(* Schneider Machine Expert - Basic project usine, file version 2.8.0.0 *)
(* ProjectInformations: Name=Nouveau projet *)

HARDWARE
  Cpu 0: TM221M16R/G
  ModuleExtensionObject 0: TM3AQ4/G
  EthernetConfiguration: NetworkName=M221, IpAllocationMode=FixedAddress, IpAddress=0.0.0.0, SubnetMask=0.0.0.0
  SerialLineConfiguration: Baud=Baud19200, Parity=ParityEven, DataBits=DataBits8, StopBits=StopBits1, PhysicalMedium=PhysicalMediumRs485, TransmissionMode=TransmissionModeModbusRtu, SlaveId=1, Addressing=SlaveAddressing
  MastTask: UsePeriodScanMode=false, PeriodScan=100
  FastTask: Period=255
  CpuBehavior: StartingMode=StartAsPreviousState, AutoSaveRamOnEeprom=true, WatchdogPeriod=250

SYMBOLS  (address, symbol, comment, settings)
  %M0       M1
  %M1       M2
  %M3       LP
  %M4       SP
  %M5       TIME
  %M6       M
  %M7       H
  %M8       MODE_AUTO
  %M9       MARCHE_DES_MACHINE
  %M10      SS
  %S6       SB_TB1S  "Base de temps de 1 s générée par une horloge interne"
  %C0         [Preset=5]
  %C1         [Preset=5]
  %C2         [Preset=4]
  %I0.0     COURANT_M_1
  %I0.1     COURANT_M_2
  %I0.2     COURANT_M_3
  %I0.3     BP
  %I0.4     BP_MARCHE
  %I0.5     BP_STOP
  %I0.6     BP_AUTO
  %I0.7     BP_AUTO_S
  %Q0.0     MACHINE_R
  %Q0.1     MACHINE_B
  %Q0.2     MOTEUR

POU cable machine
  (* SectionNumber=1 *)

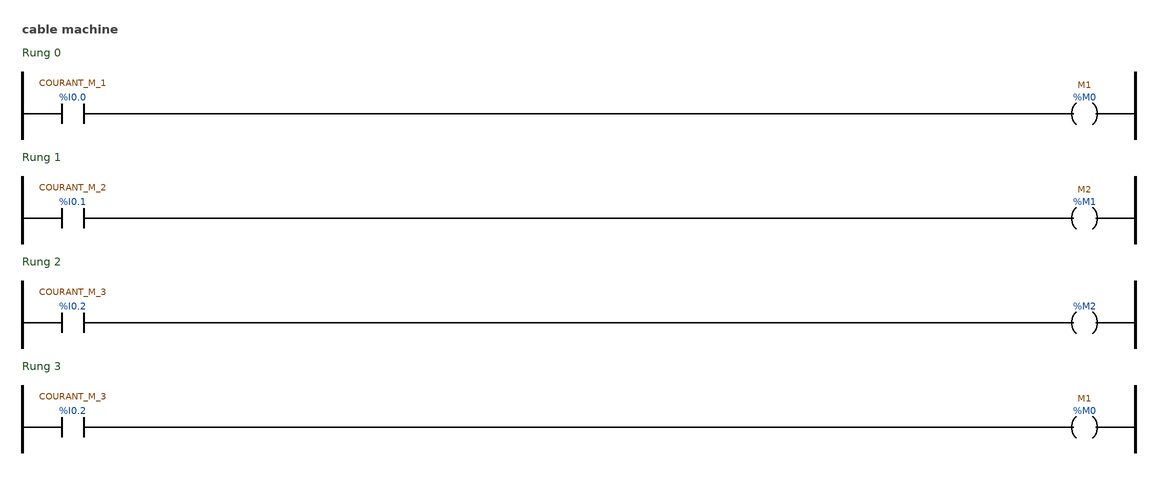

// Rung 0
  LD %I0.0                (* COURANT_M_1 *)
  ST %M0                  (* M1 *)
  // as ST:
  //   M1 := COURANT_M_1;

// Rung 1
  LD %I0.1                (* COURANT_M_2 *)
  ST %M1                  (* M2 *)
  // as ST:
  //   M2 := COURANT_M_2;

// Rung 2
  LD %I0.2                (* COURANT_M_3 *)
  ST %M2
  // as ST:
  //   %M2 := COURANT_M_3;

// Rung 3
  LD %I0.2                (* COURANT_M_3 *)
  ST %M0                  (* M1 *)
  // as ST:
  //   M1 := COURANT_M_3;

POU régulation
  (* SectionNumber=2 *)

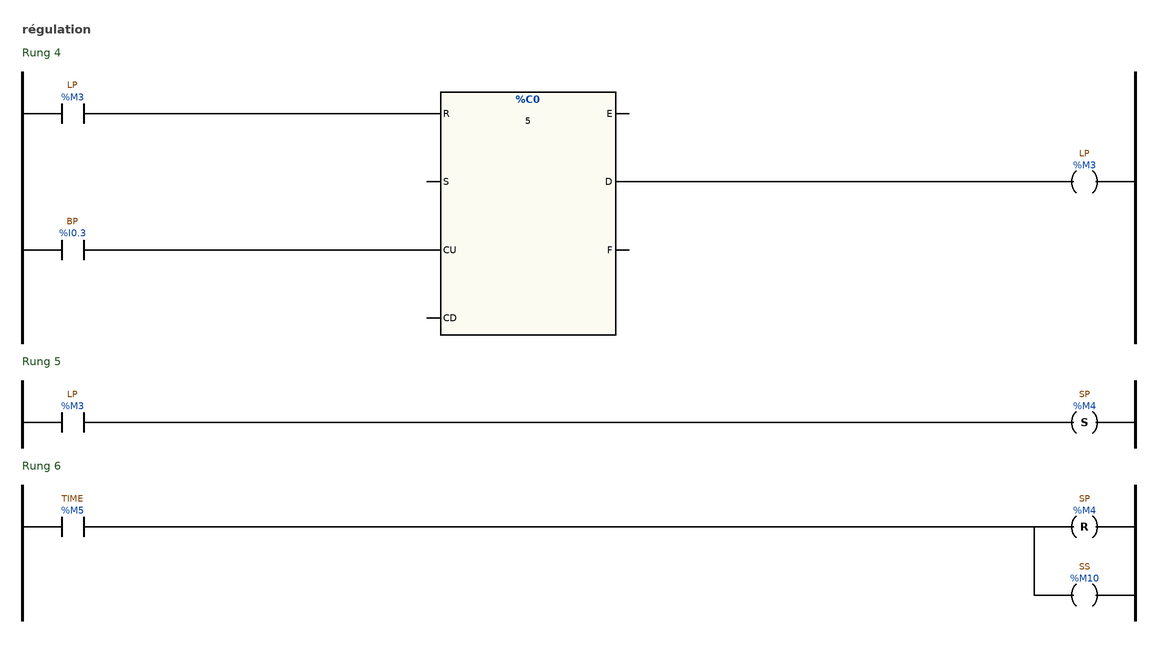

// Rung 4
  BLK %C0
  LD %M3                  (* LP *)
  R
  LD %I0.3                (* BP *)
  CU
  OUT_BLK
  LD D
  ST %M3                  (* LP *)
  END_BLK
  // as ST:
  //   %C0(R := LP, CU := BP);
  //   LP := %C0.D;

// Rung 5
  LD %M3                  (* LP *)
  S %M4                   (* SP *)
  // as ST:
  //   IF LP THEN SP := TRUE; END_IF;

// Rung 6
  LD %M5                  (* TIME *)
  R %M4                   (* SP *)
  ST %M10                 (* SS *)
  // as ST:
  //   IF TIME THEN SP := FALSE; END_IF;
  //   SS := TIME;

POU timer
  (* SectionNumber=3 *)

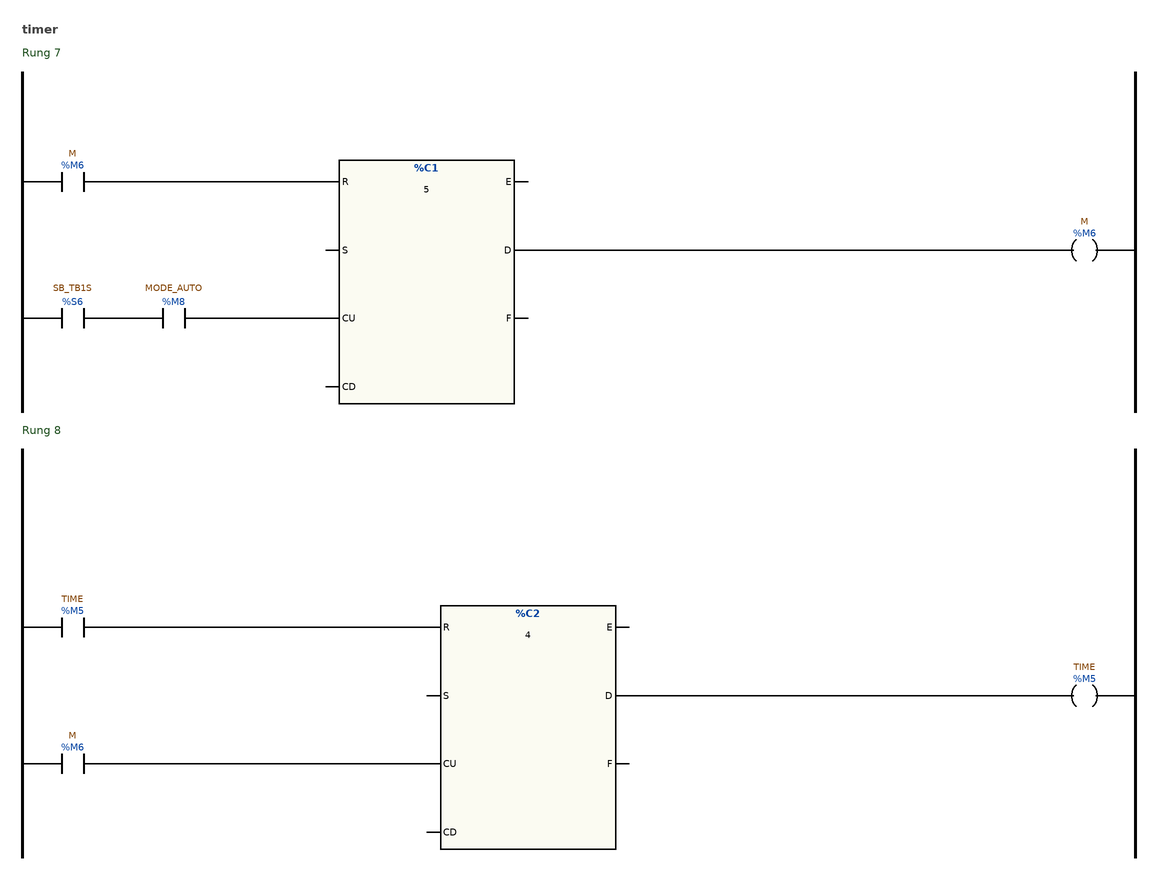

// Rung 7
  BLK %C1
  LD %M6                  (* M *)
  R
  LD %S6                  (* SB_TB1S *)
  AND %M8                 (* MODE_AUTO *)
  CU
  OUT_BLK
  LD D
  ST %M6                  (* M *)
  END_BLK
  // as ST:
  //   %C1(R := M, CU := SB_TB1S AND MODE_AUTO);
  //   M := %C1.D;

// Rung 8
  BLK %C2
  LD %M5                  (* TIME *)
  R
  LD %M6                  (* M *)
  CU
  OUT_BLK
  LD D
  ST %M5                  (* TIME *)
  END_BLK
  // as ST:
  //   %C2(R := TIME, CU := M);
  //   TIME := %C2.D;

POU start machine
  (* SectionNumber=4 *)

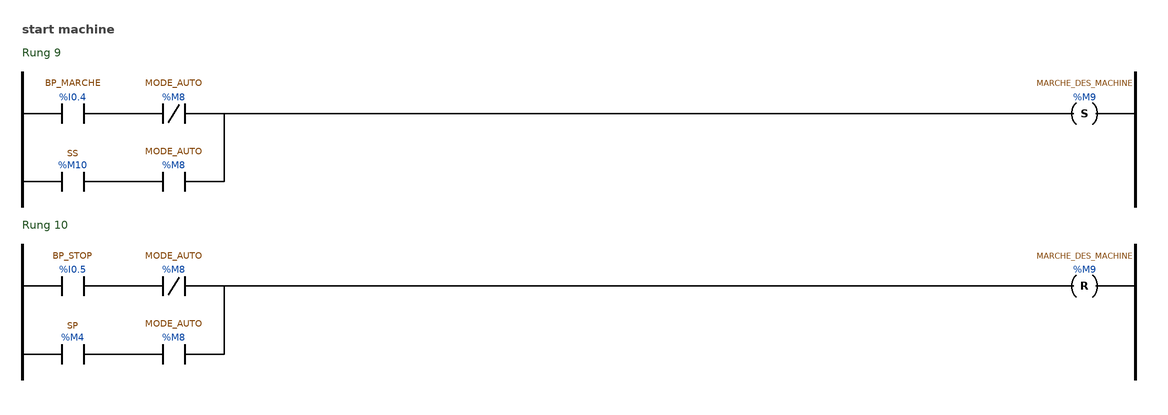

// Rung 9
  LD %I0.4                (* BP_MARCHE *)
  ANDN %M8                (* MODE_AUTO *)
  OR( %M10                (* SS *)
  AND %M8                 (* MODE_AUTO *)
  )
  S %M9                   (* MARCHE_DES_MACHINE *)
  // as ST:
  //   IF BP_MARCHE AND NOT MODE_AUTO OR SS AND MODE_AUTO THEN MARCHE_DES_MACHINE := TRUE; END_IF;

// Rung 10
  LD %I0.5                (* BP_STOP *)
  ANDN %M8                (* MODE_AUTO *)
  OR( %M4                 (* SP *)
  AND %M8                 (* MODE_AUTO *)
  )
  R %M9                   (* MARCHE_DES_MACHINE *)
  // as ST:
  //   IF BP_STOP AND NOT MODE_AUTO OR SP AND MODE_AUTO THEN MARCHE_DES_MACHINE := FALSE; END_IF;

POU mode auto
  (* SectionNumber=5 *)

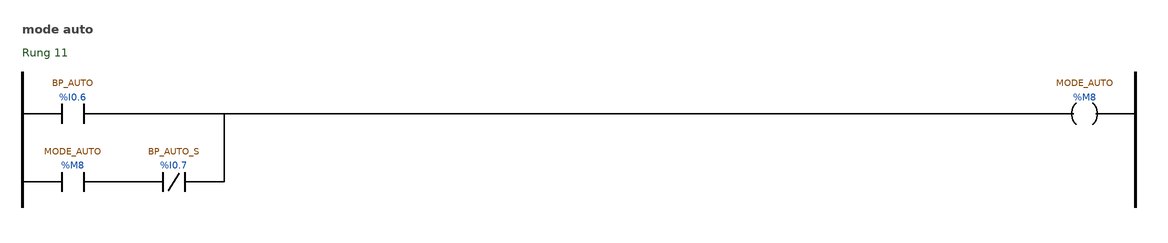

// Rung 11
  LD %I0.6                (* BP_AUTO *)
  OR( %M8                 (* MODE_AUTO *)
  ANDN %I0.7              (* BP_AUTO_S *)
  )
  ST %M8                  (* MODE_AUTO *)
  // as ST:
  //   MODE_AUTO := BP_AUTO OR MODE_AUTO AND NOT BP_AUTO_S;

POU Nouveau POU
  (* SectionNumber=0 *)

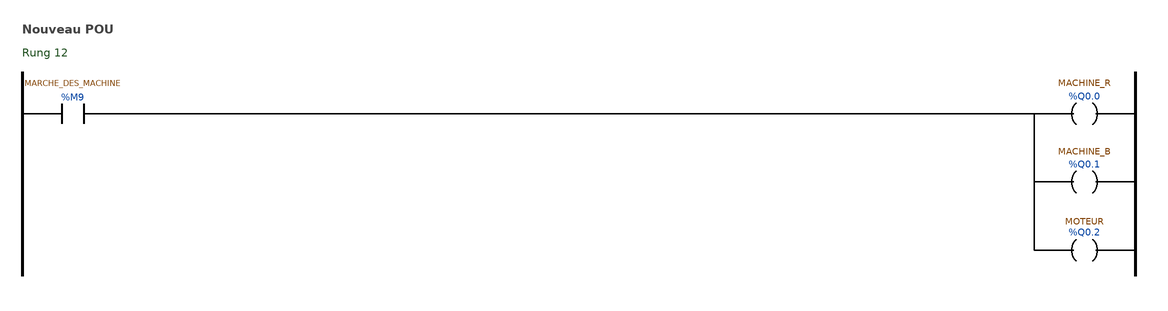

// Rung 12
  LD %M9                  (* MARCHE_DES_MACHINE *)
  ST %Q0.0                (* MACHINE_R *)
  ST %Q0.1                (* MACHINE_B *)
  ST %Q0.2                (* MOTEUR *)
  // as ST:
  //   MACHINE_R := MARCHE_DES_MACHINE;
  //   MACHINE_B := MARCHE_DES_MACHINE;
  //   MOTEUR := MARCHE_DES_MACHINE;
